// TIA Portal V18 export
// export: Created 2026-01-09T11:23:38.3957203Z, ExportSetting WithDefaults, DisplayName Totally Integrated Automation Portal, DisplayVersion V18 Update 5, DisplayName TIA Portal Openness, DisplayVersion V18 Update 5, DisplayName TIA Portal Teamcenter Gateway, DisplayVersion V18, DisplayName TIA Portal Version Control Interface, DisplayVersion V18, DisplayName SINAMICS Startdrive Advanced, DisplayVersion V18 SP2 Update 1, DisplayName SINAMICS Startdrive G110M, G120, G120C, G120D, G120P, G115D, DisplayVersion V18 SP2 Update 1, DisplayName SINAMICS Startdrive G130, G150, S120, S150, SINAMICS MV, S210, G220, S200, DisplayVersion V18 SP2 Update 1, DisplayName STEP 7 Professional, DisplayVersion V18 Update 5, DisplayName STEP 7 Safety, DisplayVersion V18, DisplayName WinCC Professional, DisplayVersion V18 Update 5
Screen "710 Recipe"  1280x800, Number=710, Template=07Parameter
  ScreenLayer "Layer_0"
    Button "btnMenu3" at 256,725 size 128x75  Mode=Text, StyleItem=BtnNormal20
    Button "btnMenu4" at 384,725 size 128x75  Mode=Text, StyleItem=BtnNormal20
    Button "btnMenu5" at 512,725 size 128x75  Mode=Text, StyleItem=BtnNormal20
    Button "btnMenu6" at 768,725 size 128x75  Mode=Text, StyleItem=BtnNormal20
    Button "btnMenu5_1" at 640,725 size 128x75  Mode=Text, StyleItem=BtnNormal20
    Button "btnMenu6_1" at 896,725 size 128x75  Mode=Text, StyleItem=BtnNormal20
    Button "btnMenu3_1" at 128,725 size 128x75  Mode=Text, StyleItem=BtnNormal20
    Button "btnMenu6_2" at 1152,725 size 128x75  Mode=Text, StyleItem=BtnNormal20
